PROGRAM Main
VAR
	fbKL6581			:	FB_KL6581;
	fbsearch 			:	FB_EnOcean_Search;
	//fbRecGeneric		: 	FB_Rec_Generic;
	readTemp			: 	readTemp2;
	whichSwitch			:	switch2;
	contactSensor1		: 	contact;
	contactSensor2		:	contact;
	
    temp			: 	REAL;
	humitity 			: 	REAL;
	switchNR			: 	INT;
	contact1			: 	BOOL;
	contact2			:	BOOL;
	tempError			:	BOOL;
	humitityError		: 	BOOL;
END_VAR

JsonEncode();

// Init
fbKL6581(bInit := TRUE, stKL6581_in := GVL_EnOcean.stKL6581Input, stKL6581_out := GVL_EnOcean.stKL6581Output);
GVL_EnOcean.stKL6581 := fbKL6581.str_KL6581;
fbsearch(bStart := TRUE, str_KL6581 := GVL_EnOcean.stKL6581, byNode := 0);

//link sensors aan POU
readTemp(sensorID := 92351965);
whichswitch(sensorID := 4277441636);
contactSensor1(sensorID := 84246605);
contactSensor2(sensorID := 84246605);

// IF sensor value changes
IF didSensorChange(readTemp := readTemp, whichSwitch := whichSwitch) THEN
	temp := readTemp.tempOutput;
	humitity := readTemp.humitityOut;
	switchNR := whichSwitch.switchNR;
	contact1 := contactSensor1.contact;
	contact2 := contactSensor2.contact;
	mqttconn();
END_IF
	
// handle exceptions	

IF temp < 20 OR temp > 40 THEN
	tempError := TRUE;
END_IF

IF humitity < 40 OR humitity > 60 THEN
	humitityError := TRUE;
END_IF

(*
IF switchNR <> 0 THEN
	IF switchNR = 2 THEN
		<handle switch>
	END_IF
END_IF
*)

(*
Sensor IDs:
Temp+vochtig ==> 92351965 : ar_value[1] = temp, ar_value[2] = vochtig
schakelaar ==> 4277441636 : ar_value[3]
raamcontact1 ==> 84246605 : ar_value[3]
raamcontact2 ==> 84246441: ar_value[3]




*)

END_PROGRAM

(* stored: Version 1.1.0.1, ProductVersion 3.1.4022.17
   POU Main: Id {39b8f405-16cb-4a36-9c9e-2b9b67c73480}, SpecialFunc None *)
